Universal Robots PolyScope program: Password_Move_UR.urp

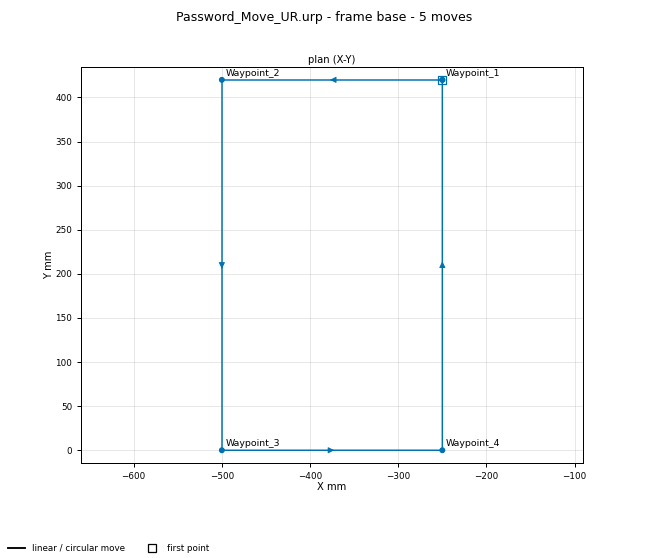
[picture p0: tool path of Password_Move_UR.urp in frame base, 5 of 5 moves have a stored position in this frame; points joined in program order, loops and branches not executed]
Program PASSWORD move (installation=password directory=/programs/usbdisk createdIn=5.11.9 lastSavedIn=5.13.0 robotSerialNumber=20205001148)
Calibrated DH parameters: a=[0.000006, -0.588386, 0.024864, -0.000008, 0.000016, 0]; d=[0.180784, -42.502966, -480.259695, 522.93681, 0.119862, 0.115521]; alpha=[1.570208, -0.003949, 0.001092, 1.570374, -1.570321, 0]; deltaTheta=[0, 0.277877, 4.390974, 1.614336, -0.000001, 0]
InitVariablesNode
Robot Program (runOnlyOnce=false)
  MoveJ speed 60 deg/s, acceleration 80 deg/s^2 (useActiveTCP=true) feature=Base
    Waypoint Waypoint_1: TCP in base x=-250 y=420 z=0 mm, rx=2.2038 ry=-2.2038 rz=-0.0385 rad; joints [-76.208, -53.575, 90.582, 52.443, 87.821, -75.986] deg; TCP offset x=0 y=0 z=167.69 mm, rx=0 ry=0 rz=0 rad
  Loop Counting (count=30) loopVariable(name=Loop_1)
    MoveL speed 250 mm/s, acceleration 1200 mm/s^2 (useActiveTCP=true) feature=Base
      Wait Sleep waitTime=5
      Waypoint Waypoint_2: motionParameters(nextMotionTime=1); TCP in base x=-500 y=420 z=0.003 mm, rx=2.2039 ry=-2.2037 rz=-0.0385 rad; joints [-52.506, -32.453, 50.371, 70.796, 88.096, -52.389] deg; TCP offset x=0 y=0 z=167.69 mm, rx=0 ry=0 rz=0 rad
      Waypoint Waypoint_3: motionParameters(nextMotionTime=1); TCP in base x=-500 y=0 z=0 mm, rx=2.2038 ry=-2.2038 rz=-0.0385 rad; joints [-15.8, -53.041, 89.16, 51.889, 89.222, -15.577] deg; TCP offset x=0 y=0 z=167.69 mm, rx=0 ry=0 rz=0 rad
      Waypoint Waypoint_4: motionParameters(nextMotionTime=1); TCP in base x=-250.006 y=0.005 z=-0.021 mm, rx=2.2038 ry=-2.2038 rz=-0.0383 rad; joints [-33.702, -81.37, 134.186, 35.453, 88.741, -33.397] deg; TCP offset x=0 y=0 z=167.69 mm, rx=0 ry=0 rz=0 rad
      Waypoint Waypoint_1: motionParameters(nextMotionTime=1); TCP in base x=-250 y=420 z=0 mm, rx=2.2038 ry=-2.2038 rz=-0.0385 rad; joints [-76.208, -53.575, 90.582, 52.443, 87.821, -75.986] deg; TCP offset x=0 y=0 z=167.69 mm, rx=0 ry=0 rz=0 rad
  Halt
